% RSLogix 500 project 7.2.RSS, saved by version 8.30.00.16 %
PROJECT "UNTITLED"    % processor: Bul.1763 MicroLogix 1100 Series B %

PROGRAM FILES
  LAD 2   7 rungs

DATA FILES
  O0 OUTPUT  4 elements
  I1 INPUT  6 elements
  S2 STATUS  66 elements
  B3 BINARY  1 elements
  T4 TIMER  3 elements
  C5 COUNTER  1 elements
  R6 CONTROL  1 elements
  N7 INTEGER  1 elements
  F8 FLOAT  1 elements

LADDER 2
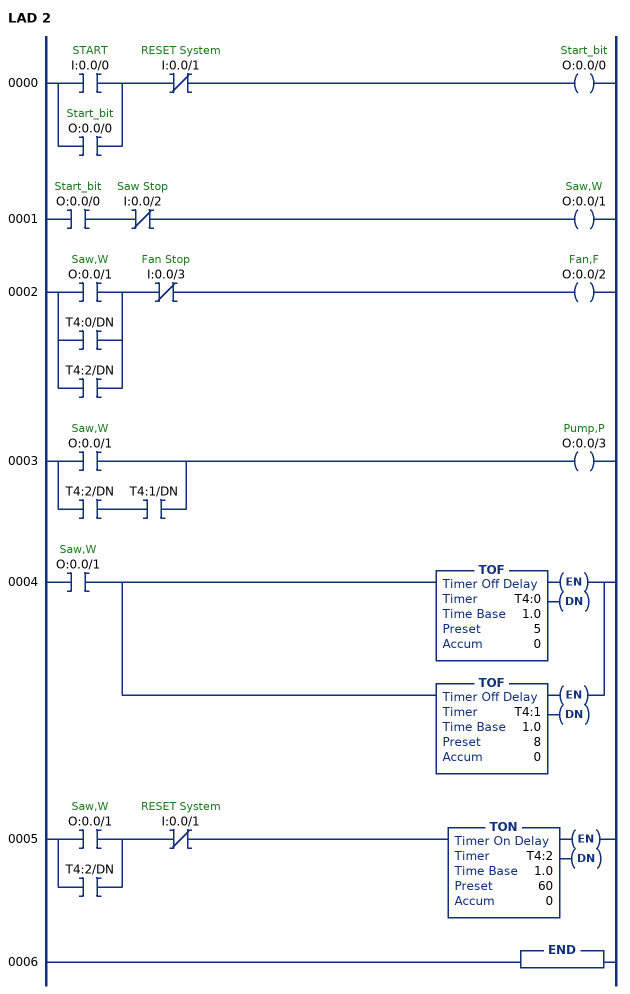
% Rung: 0 %
SOR BST XIC I:0.0/0 NXB XIC O:0.0/0 BND XIO I:0.0/1 OTE O:0.0/0 EOR
%   I:0.0/0  "START" %
%   O:0.0/0  "Start_bit" %
%   I:0.0/1  "RESET System" %
% Rung: 1 %
SOR XIC O:0.0/0 XIO I:0.0/2 OTE O:0.0/1 EOR
%   O:0.0/0  "Start_bit" %
%   I:0.0/2  "Saw Stop" %
%   O:0.0/1  "Saw,W" %
% Rung: 2 %
SOR BST XIC O:0.0/1 NXB BST XIC T4:0/DN NXB XIC T4:2/DN BND BND XIO I:0.0/3 OTE O:0.0/2 EOR
%   O:0.0/1  "Saw,W" %
%   I:0.0/3  "Fan Stop" %
%   O:0.0/2  "Fan,F" %
% Rung: 3 %
SOR BST XIC O:0.0/1 NXB XIC T4:2/DN XIC T4:1/DN BND OTE O:0.0/3 EOR
%   O:0.0/1  "Saw,W" %
%   O:0.0/3  "Pump,P" %
% Rung: 4 %
SOR XIC O:0.0/1 BST TOF T4:0 1.0 5 0 NXB TOF T4:1 1.0 8 0 BND EOR
%   O:0.0/1  "Saw,W" %
% Rung: 5 %
SOR BST XIC O:0.0/1 NXB XIC T4:2/DN BND XIO I:0.0/1 TON T4:2 1.0 60 0 EOR
%   O:0.0/1  "Saw,W" %
%   I:0.0/1  "RESET System" %
% Rung: 6 %
SOR END EOR

DATA TABLE (non-zero values as saved)
DATA T4
% .PRE .ACC %
% T4:0 % 5 0
% T4:1 % 8 0
% T4:2 % 60 0
